{attribute addProperty BoxType "EJ3255-0000-0023"}
{attribute addProperty Id "AI_Standard_ChannelAT %I*ARRAY[0..4] OF AI_Standard_Channel_087F71C7160200WcStateAT %I*WcState_F855686C1620InfoDataAT %I*InfoData_BC63D37F80100"}
{attribute addProperty CRC "2220818549"}
{attribute addProperty SizeInBites "256"}
{attribute addProperty SizeInBytes "32"}
TYPE EJ3255_A08AFE1A :
STRUCT
	{attribute addProperty Name "AI_Standard_Channel"}
	AI_Standard_Channel : ARRAY[0..4] OF AI_Standard_Channel_087F71C7;
	{attribute addProperty Name "WcState"}
	WcState : WcState_F855686C;
	{attribute addProperty Name "InfoData"}
	InfoData : InfoData_BC63D37F;
END_STRUCT
END_TYPE

(* stored: Version 1.2.0.0, ProductVersion 3.1.4024.9
   DUT EJ3255_A08AFE1A: Id {484912fc-635b-4675-9b8e-5fa07422b1c4} *)
